FUNCTION_BLOCK CNV_CTRL (* Composite Function Block Type *)
  (* Standard: 61499-2 *)
  (* Version 0.2, 2003-12-05, JHC, Rockwell Automation, Renamed from NEWCOMPFB. *)
  (* Version 0.1, 2002-01-08, JHC, Rockwell Automation, Added DLY FB as example. *)
  (* Version 0.0, 2000-05-27, JHC, Rockwell Automation *)
  (* Compiler header: package fb.rt.template; *)
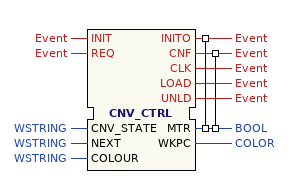
  EVENT_INPUT
    INIT; (* Initialization Request *)
    REQ; (* Normal Execution Request *)
  END_EVENT
  EVENT_OUTPUT
    INITO WITH MTR; (* Initialization Confirm *)
    CNF WITH MTR; (* Execution Confirmation *)
    CLK;
    LOAD;
    UNLD;
  END_EVENT
  VAR_INPUT
    CNV_STATE : WSTRING;
    NEXT : WSTRING;
    COLOUR : WSTRING;
  END_VAR
  VAR_OUTPUT
    MTR : BOOL; (* Output event qualifier *)
    WKPC : COLOR;
  END_VAR
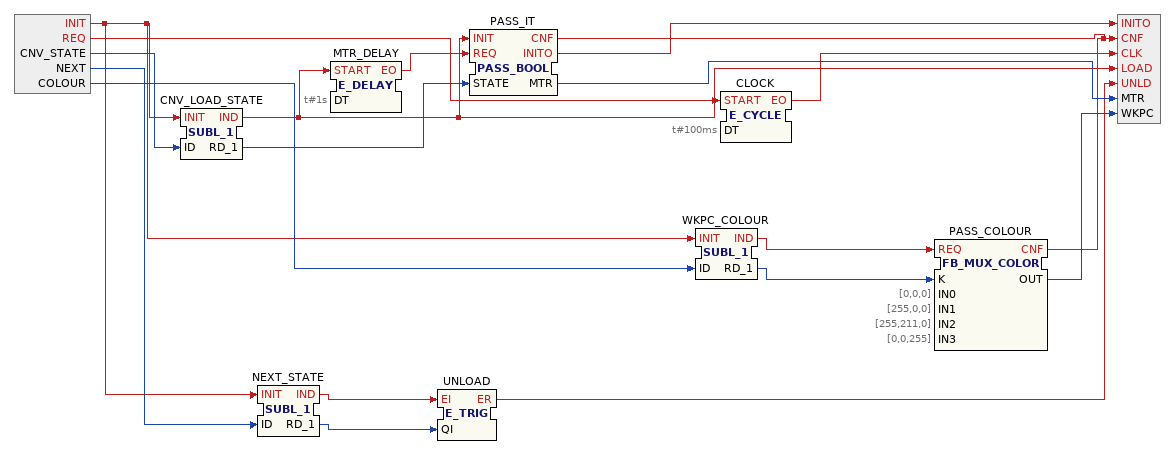
  FBS
    NEXT_STATE : SUBL_1;
    UNLOAD : E_TRIG;
    CLOCK : E_CYCLE(DT := t#100ms);
    PASS_COLOUR : FB_MUX_COLOR(IN0 := [0,0,0], IN1 := [255,0,0], IN2 := [255,211,0], IN3 := [0,0,255]);
    WKPC_COLOUR : SUBL_1;
    MTR_DELAY : E_DELAY(DT := t#1s);
    CNV_LOAD_STATE : SUBL_1;
    PASS_IT : PASS_BOOL;
  END_FBS
  EVENT_CONNECTIONS
    INIT TO NEXT_STATE.INIT;
    NEXT_STATE.IND TO UNLOAD.EI;
    CLOCK.EO TO CLK;
    REQ TO CLOCK.START;
    UNLOAD.ER TO UNLD;
    PASS_COLOUR.CNF TO CNF;
    INIT TO WKPC_COLOUR.INIT;
    WKPC_COLOUR.IND TO PASS_COLOUR.REQ;
    INIT TO CNV_LOAD_STATE.INIT;
    CNV_LOAD_STATE.IND TO LOAD;
    CNV_LOAD_STATE.IND TO MTR_DELAY.START;
    CNV_LOAD_STATE.IND TO PASS_IT.INIT;
    MTR_DELAY.EO TO PASS_IT.REQ;
    PASS_IT.CNF TO CNF;
    PASS_IT.INITO TO INITO;
  END_CONNECTIONS
  DATA_CONNECTIONS
    NEXT_STATE.RD_1 TO UNLOAD.QI;
    NEXT TO NEXT_STATE.ID;
    PASS_COLOUR.OUT TO WKPC;
    WKPC_COLOUR.RD_1 TO PASS_COLOUR.K;
    COLOUR TO WKPC_COLOUR.ID;
    CNV_STATE TO CNV_LOAD_STATE.ID;
    CNV_LOAD_STATE.RD_1 TO PASS_IT.STATE;
    PASS_IT.MTR TO MTR;
  END_CONNECTIONS
END_FUNCTION_BLOCK
